// TIA Portal V20 export
TYPE "LBP_typeInternal4"
TITLE = Internal data type for basic program / Type de données interne pour programme de base
// Data type only for internal use in the basic program / Type de données réservé à l'utilisation interne dans le programme de base
   STRUCT
      Handwheels : Array[1..6] of Struct
         active : Bool;
         recent : Bool;
         stopped : Bool;
         pulses : Int;
      END_STRUCT;
   END_STRUCT;
END_TYPE
